FUNCTION_BLOCK Q_ListItem (* Command change list item ( Part 6 - F.42 ) *)
  (* Standard: ISO 11783-6; Description: Copyright (c) 2022 HR Agrartechnik GmbH This program and the accompanying materials are made available under the terms of the Eclipse Public License 2.0 which is available at https://www.eclipse.org/legal/epl-2.0/ SPDX-License-Identifier: EPL-2.0 see Description Tab *)
  (* Version 1.0, 2022-07-08, Franz Höpfinger, HR Agrartechnik GmbH *)
  PACKAGE isobus::UT::Q;
  IMPORT isobus::UT::Q::const::IDs::ID_NULL;
  (* Documentation:
  Command change list item ( Part 6 - F.42 )
   This command is used to change a list item in an Input List, Output List, Animation, or External Object Definition object.
   Valid values for u16ObjId (the list object)
   A list item Object ID is valid if it falls within one of the following ISO 11783-6 ID ranges (Annex F.42):
    - InputListField: 10000 – 10999
   - OutputListObject: 37000 – 37999 (VT version 4 and later)
   - AnimationObject: 44000 – 44999 (VT version 5 and later)
   - ExternalObjectDef: 41000 – 41999 (VT version 5 and later)
    ID_NULL (65535) is not a command target but can be used in INIT to deactivate the FB. Any ID outside these ranges is invalid for commanding.
   Valid values for u16NewObjId (the new list item)
   Annex F.42 permits any Object ID as the new list item — the item simply points to that object — or FFFF16 (ID_NULL) to set an empty item. The validity of the new Object ID is verified by the VT and reported back in the F.43 response (bit 2 = Invalid New List Item Object ID).
   Activate / Deactivate
   The FB is deactivated by default. It becomes active when INIT provides a valid list item Object ID. Sending INIT with ID_NULL (65535) deactivates the FB again. This toggle can be repeated arbitrarily.
    - INIT + ID_NULL (65535): FB deactivated, STATUS="DEACTIVATED", s16result=VT_E_DEACTIVATED (-40)
   - INIT + valid list item ID: FB activated, STATUS="initialized", s16result=VT_E_NO_ERR (0). If a REQ was buffered before, it is executed immediately.
   - INIT + invalid ID: STATUS="ERROR: Invalid Object ID (not a list item object)", s16result=VT_E_INVALID_OBJECT_ID (-132)
    REQ Handling
    - REQ before any INIT: Buffered, STATUS="Buffered: INIT not yet completed", s16result=VT_E_NOT_READY (-131)
   - REQ while deactivated (INIT came with NULL or invalid ID): STATUS shows the actual deactivation reason, s16result=VT_E_DEACTIVATED (-40) or VT_E_INVALID_OBJECT_ID (-132)
   - REQ while active: Command sent to VT, result reflected in CNF
    param[in] {objectID, uint16_t}
   Object ID of a list/input/object. Use ID_NULL (65535) to deactivate the FB. Use a valid list item object ID to activate.
   param[in] {listIndex, uint8_t}
   List index (-> see list)
   param[in] {newObjectID, uint16_t}
   New object ID or 0xFFFF to set empty
   Return Values (s16result):
   int16_t
    - VT_E_NO_ERR (0) - OK
   - VT_E_DEACTIVATED (-40) - FB deactivated (INIT received with ID_NULL)
   - VT_E_INVALID_OBJECT_ID (-132) - Object ID is invalid (not a list item object)
   - VT_E_NOT_READY (-131) - Buffered: INIT not yet completed
   - VT_E_OVERFLOW (-6) - buffer overflow
   - VT_E_NOACT (-8) - Command not possible in current state
   - VT_E_NO_INSTANCE (-21) - No VT client available
   - VT_E_ISO_INSTANCE_INVALID (-129) - Identifier for instance (connection) invalid
   - VT_E_NOT_ALIVE (-130) - Identifier for instance valid, but VT Dead.
    Instanz-Eindeutigkeit (Instance Uniqueness)
   Dieser Baustein erfordert Instanz-Eindeutigkeit bezüglich des Paares (u16ObjId, u8ListIndex). Es darf im gesamten Programm nur eine Instanz von Q_ListItem für denselben Listeneintrag existieren. u8ListIndex wird bei INIT eingelesen — eine zweite Instanz auf dieselbe Listen-Objekt-ID und denselben Listen-Index wird bei INIT deaktiviert (STATUS = "This objID is already in use").
  *)
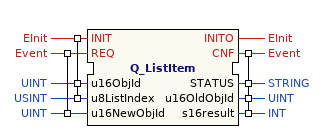
  EVENT_INPUT
    INIT : EInit WITH u16ObjId, u8ListIndex; (* Service Initialization *)
    REQ WITH u16NewObjId; (* Service Request *)
  END_EVENT
  EVENT_OUTPUT
    INITO : EInit; (* Initialization Confirm *)
    CNF WITH STATUS, s16result, u16OldObjId; (* Confirmation of Requested Service *)
  END_EVENT
  VAR_INPUT
    u16ObjId : UINT := ID_NULL; (* Object ID *)
    u8ListIndex : USINT; (* List index (-> see list) *)
    u16NewObjId : UINT := ID_NULL; (* New object ID or 0xFFFF to set empty *)
  END_VAR
  VAR_OUTPUT
    STATUS : STRING; (* Service Status *)
    u16OldObjId : UINT; (* Old object ID or 0xFFFF to set empty *)
    s16result : INT; (* retval see description *)
  END_VAR
END_FUNCTION_BLOCK
